PROGRAM MAIN
VAR
	asd: BOOL;
	doubl: BOOL;
END_VAR

asd := doubl;

END_PROGRAM

(* stored: Version 1.1.0.1, ProductVersion 3.1.4024.10
   POU MAIN: Id {c05d75f6-1e14-47e5-98de-612ecc680255}, SpecialFunc None *)
